Staubli VAL3: Prise.pgx

program Prise(point x_pPoint (dimensions=1))
begin
  movej(appro(x_pPoint,trAppro),tPince,mRapide)
  open(tPince)
  movel(x_pPoint,tPince,mLent)
  close(tPince)
  movel(appro(x_pPoint,trAppro),tPince,mLent)
end
